// TIA Portal V19 export
TYPE "type_u3ToXyz"
// stored: Access Published, Namespace Unit3
   STRUCT
      deliver : "Unit3.type_u3RequestData";
      recieve : "Unit3.type_u3ResponsetData";
   END_STRUCT;
END_TYPE
